// TIA Portal V16 export
// export: Created 2024-12-03T15:41:43.2889694Z, ExportSetting WithDefaults, DisplayName Totally Integrated Automation Portal, DisplayVersion V16 Update 6, DisplayName TIA Portal Version Control Interface, DisplayVersion V16 Update 2, DisplayName TIA Portal Openness, DisplayVersion V16 Update 6, DisplayName TIA Portal Teamcenter Gateway, DisplayVersion V16, DisplayName SINAMICS Startdrive Advanced, DisplayVersion V16 Update 5, DisplayName SINAMICS Startdrive G130, G150, S120, S150, SINAMICS MV, S210, DisplayVersion V16 Update 5, DisplayName SINAMICS Startdrive G110M, G120, G120C, G120D, G120P, G115D, DisplayVersion V16 Update 5, DisplayName STEP 7 Professional, DisplayVersion V16 Update 6, DisplayName STEP 7 Safety, DisplayVersion V16, DisplayName WinCC Advanced / Unified PC, DisplayVersion V16 Update 6
FUNCTION_BLOCK "Intersection_Controller_FB"   // FB30, SCL
{ S7_Optimized_Access := 'TRUE' }
VERSION : 0.1
// stored: AutoNumber true, IsIECCheckEnabled false, IsRetainMemResEnabled false, MemoryReserve 100, SetENOAutomatically false, UDAEnableTagReadback false
   VAR_INPUT
      I_con_upstream_north : Bool := TRUE;
      I_con_upstream_east : Bool := TRUE;
      I_con_upstream_south : Bool := TRUE;
      I_con_upstream_west : Bool := TRUE;
      I_Conv_North : "Conveyor_UDT";
      I_Conv_East : "Conveyor_UDT";
      I_Conv_South : "Conveyor_UDT";
      I_Conv_West : "Conveyor_UDT";
      I_Settings : "Intersection";
      I_AutoSent : Bool;
   END_VAR
   VAR_OUTPUT
      O_Empty_Flag : Bool;
   END_VAR
   VAR_IN_OUT
      IO_Conv_1 : "Conveyor_UDT";
      IO_Conv_2 : "Conveyor_UDT";
      IO_Transfer : "TransferUnitUpDown";
   END_VAR
   VAR
      Transfer : "ZPA_TransferUnit_Controller";
   END_VAR
   VAR RETAIN
      settings { S7_SetPoint := 'True'} : "Intersection";
   END_VAR
   VAR
      Empty { S7_SetPoint := 'True'} : "SmartBool";
   END_VAR
   VAR_TEMP
      T_Zone : "ZoneInfo";
      T_appstate : "ApplicationState_UDT";
      T_DownStream : "Conveyor_UDT";
      T_Upstream : "Conveyor_UDT";
      T_SendingConveyor : "Conveyor_UDT";
      T_ReceiveConveyor : "Conveyor_UDT";
      T_ReceivePosition : Int;
      T_InvalidSettings : Bool;
      T_Dummy : Bool;
      T_ConnectUpstream : Bool;
   END_VAR
BEGIN
   REGION INit temps

       #T_Zone := "ApplicationState_DB".ZoneNames[#IO_Conv_1.Zone];
       #T_appstate := "ApplicationState_DB".Appstate[#T_Zone.AppStateIndex];

       #T_DownStream := "CONV_DB".empty;
       #T_Upstream := "CONV_DB".empty;
       #T_SendingConveyor := "CONV_DB".empty;
       #T_ReceiveConveyor := "CONV_DB".empty;

   END_REGION

   REGION INIT NAMES

       IF #IO_Conv_1.Name = '' THEN
           #IO_Conv_1.Name := "buildObjectName"(I_Symbolname := GetSymbolName(variable:=#IO_Conv_1, size:=60));
       END_IF;

       IF #IO_Conv_2.Name = '' THEN
           #IO_Conv_2.Name := "buildObjectName"(I_Symbolname := GetSymbolName(variable := #IO_Conv_2, size := 60));
       END_IF;
   END_REGION

   REGION Allow new settings

       IF (#IO_Conv_1.Status.Empty
           AND #IO_Conv_2.Status.Empty) THEN //OR #settings.DownstreamIndex = 0 THEN
           #settings := #I_Settings;
       END_IF;

       #T_ReceivePosition := #settings.ReceivePosition;

   END_REGION

   REGION DownStream Selecotor

       CASE #settings.DownstreamIndex OF
           "North":
               #T_DownStream := #I_Conv_North  ;
           "East":
               #T_DownStream := #I_Conv_East ;
           "South":
               #T_DownStream := #I_Conv_South ;
           "West":
               #T_DownStream := #I_Conv_West ;
       END_CASE;

   END_REGION

   REGION Upstream selector

       #T_ConnectUpstream := FALSE;

       CASE #settings.UpstreamIndex OF
           "North":
               #T_Upstream := #I_Conv_North;
               #T_ConnectUpstream := #I_con_upstream_north;
           "East":
               #T_Upstream := #I_Conv_East;
               #T_ConnectUpstream := #I_con_upstream_east;
           "South":
               #T_Upstream := #I_Conv_South;
               #T_ConnectUpstream := #I_con_upstream_south;
           "West":
               #T_Upstream := #I_Conv_West;
               #T_ConnectUpstream := #I_con_upstream_west;
       END_CASE;

   END_REGION

   REGION Init conveyors

       #IO_Conv_1.Cmd.ReadyToReceive := 0;
       #IO_Conv_1.Cmd.ReadyToSent := 0;
       #IO_Conv_1.Cmd.InvertFlow := 0;
       #IO_Conv_1.Cmd.RunAuto := 0;

       #IO_Conv_1.Status.Empty := FALSE;

       #IO_Conv_1.Status.ExecutingReceiveSequence := FALSE;
       #IO_Conv_1.Status.ExecutingSendingSequence := FALSE;
       #IO_Conv_1.Status.RequestForSending := FALSE;

       #IO_Conv_2.Cmd.ReadyToReceive := 0;
       #IO_Conv_2.Cmd.ReadyToSent := 0;
       #IO_Conv_2.Cmd.InvertFlow := 0;
       #IO_Conv_2.Cmd.RunAuto := 0;

       #IO_Conv_2.Status.Empty := FALSE;

       #IO_Conv_2.Status.ExecutingReceiveSequence := FALSE;
       #IO_Conv_2.Status.ExecutingSendingSequence := FALSE;
       #IO_Conv_2.Status.RequestForSending := FALSE;

   END_REGION

   REGION Setup conveyors

       CASE #settings.ReceiveConveyorIndex OF
           1:
               #T_ReceiveConveyor := #IO_Conv_1;
           2:
               #T_ReceiveConveyor := #IO_Conv_2;
       END_CASE;

       CASE #settings.SendingConveyorIndex OF
           1:
               #T_SendingConveyor := #IO_Conv_1;
           2:
               #T_SendingConveyor := #IO_Conv_2;
       END_CASE;


       REGION ALIGNMENT OVERRIDE
           IF #Transfer.StepNumber = 60 THEN
               #T_ReceivePosition := #settings.Algin.AlginPosition;
               CASE #settings.Algin.conveyorIndex OF
                   1:
                       #T_ReceiveConveyor.Cmd := #IO_Conv_1.Cmd;
                       #T_ReceiveConveyor.Status := #IO_Conv_1.Status;
                       #T_ReceiveConveyor.Input := #IO_Conv_1.Input;
                       #T_ReceiveConveyor.Settings := #IO_Conv_1.Settings;
                       #T_ReceiveConveyor.Encoder := #IO_Conv_1.Encoder;
                   2:
                       #T_ReceiveConveyor.Cmd := #IO_Conv_2.Cmd;
                       #T_ReceiveConveyor.Status := #IO_Conv_2.Status;
                       #T_ReceiveConveyor.Input := #IO_Conv_2.Input;
                       #T_ReceiveConveyor.Settings := #IO_Conv_2.Settings;
                       #T_ReceiveConveyor.Encoder := #IO_Conv_2.Encoder;
               END_CASE;
           END_IF;
       END_REGION

       #T_ReceiveConveyor.Cmd.InvertFlow := #settings.InverseFlowReceiving;
       #T_SendingConveyor.Cmd.InvertFlow := #settings.InverseFlowSending;

   END_REGION

   REGION ZPA transfer unit
       #T_InvalidSettings := FALSE;
       IF #settings.DownstreamIndex = 0
           OR #settings.UpstreamIndex = 0
           OR #settings.SendingConveyorIndex = 0
           OR #settings.ReceiveConveyorIndex = 0
           OR #settings.ReceivePosition = 0
           OR #settings.SendingPosition = 0 THEN
           #T_InvalidSettings := true;
       END_IF;

       IF #T_InvalidSettings THEN
           #T_ReceiveConveyor := #IO_Conv_1;
           #T_SendingConveyor := #IO_Conv_2;
           #settings.ReceivePosition := "Down";
           #settings.SendingPosition := "Up";
       END_IF;

       #Transfer(I_BuildName:=FALSE,
                 I_SentAtEnd:= #I_AutoSent,
                 I_ConnectUpstream:= #T_ConnectUpstream,
                 I_UpstreamConveyor := #T_Upstream,
                 I_DownStreamConveyor := #T_DownStream,
                 I_ReceivePosition := #T_ReceivePosition,
                 I_SendingPosition := #settings.SendingPosition,
                 I_NoEndSensor:= #settings.ReceiveNoEndSensor,
                 I_AlignAfterReceive:=#settings.Algin.active,
                 I_AlignConveyorIndex := 1, // We always the the align conveyor the receive conveyor and set the receive conveyor,
                 I_AlignSpeed:=#settings.Algin.speed,
                 I_AlignDirection:=#settings.Algin.direction,
                 I_AlignDistance:=#settings.Algin.distnace,
                 I_AlignPostition:=#settings.Algin.AlginPosition,
                 IO_ReceiveConveyor := #T_ReceiveConveyor,
                 IO_SendingConveyor := #T_SendingConveyor,
                 IO_VLV_Transfer := #IO_Transfer); 

       #T_Dummy := #T_SendingConveyor.Cmd.Direction;

   END_REGION

   REGION update conveyors with transfer unit commands

       IF #settings.ReceiveConveyorIndex <> #settings.SendingConveyorIndex THEN

           CASE #settings.ReceiveConveyorIndex OF
               1:
                   #IO_Conv_1 := #T_ReceiveConveyor;
               2:
                   #IO_Conv_2 := #T_ReceiveConveyor;
           END_CASE;

           CASE #settings.SendingConveyorIndex OF
               1:
                   #IO_Conv_1 := #T_SendingConveyor;
               2:
                   #IO_Conv_2 := #T_SendingConveyor;
           END_CASE;

       ELSE

           IF #settings.ReceiveConveyorIndex = 1 AND #settings.SendingConveyorIndex = 1 THEN

               #IO_Conv_1.Cmd.RunAuto := #T_ReceiveConveyor.Cmd.RunAuto OR #T_SendingConveyor.Cmd.RunAuto;

               IF #T_ReceiveConveyor.Status.ExecutingReceiveSequence THEN
                   #IO_Conv_1 := #T_ReceiveConveyor;
               ELSIF #T_SendingConveyor.Status.ExecutingSendingSequence THEN
                   #IO_Conv_1 := #T_SendingConveyor;
               END_IF;
           END_IF;

           IF #settings.ReceiveConveyorIndex = 2 AND #settings.SendingConveyorIndex = 2 THEN

               #IO_Conv_2.Cmd.RunAuto := #T_ReceiveConveyor.Cmd.RunAuto OR #T_SendingConveyor.Cmd.RunAuto;

               IF #T_ReceiveConveyor.Status.ExecutingReceiveSequence THEN
                   #IO_Conv_2 := #T_ReceiveConveyor;
               ELSIF #T_SendingConveyor.Status.ExecutingSendingSequence THEN
                   #IO_Conv_2 := #T_SendingConveyor;
               END_IF;
           END_IF;

       END_IF;

       REGION ALIGNMENT FUNCTION
           IF #Transfer.StepNumber = 60 THEN
               CASE #settings.Algin.conveyorIndex OF
                   1:
                       #IO_Conv_1.Cmd := #T_ReceiveConveyor.Cmd;
                       #IO_Conv_1.Input := #T_ReceiveConveyor.Input;
                       #IO_Conv_1.Status := #T_ReceiveConveyor.Status;
                       #IO_Conv_1.Encoder :=#T_ReceiveConveyor.Encoder;
                       #IO_Conv_1.Settings := #T_ReceiveConveyor.Settings;
                       #IO_Conv_2.Cmd.RunAuto := 0;
                   2:
                       #IO_Conv_2.Cmd := #T_ReceiveConveyor.Cmd;
                       #IO_Conv_2.Cmd := #T_ReceiveConveyor.Cmd;
                       #IO_Conv_2.Input := #T_ReceiveConveyor.Input;
                       #IO_Conv_2.Status := #T_ReceiveConveyor.Status;
                       #IO_Conv_2.Encoder := #T_ReceiveConveyor.Encoder;
                       #IO_Conv_2.Settings := #T_ReceiveConveyor.Settings;
                       #IO_Conv_1.Cmd.RunAuto := 0;
               END_CASE;
           END_IF;
       END_REGION

       //Empty status of conveyors must always be the same
       #IO_Conv_1.Status.Empty := #T_SendingConveyor.Status.Empty OR #T_ReceiveConveyor.Status.Empty;
       #IO_Conv_2.Status.Empty := #T_SendingConveyor.Status.Empty OR #T_ReceiveConveyor.Status.Empty;



   END_REGION

   REGION ALARMS

       #IO_Conv_1.Alarms := #T_SendingConveyor.Alarms;

       #IO_Conv_1.Alarms.BlockedReceive.Active := #T_SendingConveyor.Alarms.BlockedReceive.Active
       OR #T_ReceiveConveyor.Alarms.BlockedReceive.Active;

       #IO_Conv_1.Alarms.BlockedSending.Active := #T_SendingConveyor.Alarms.BlockedSending.Active
       OR #T_ReceiveConveyor.Alarms.BlockedSending.Active;

       #IO_Conv_1.Alarms.ToClose.Active := #T_SendingConveyor.Alarms.ToClose.Active
       OR #T_ReceiveConveyor.Alarms.ToClose.Active;

       #IO_Conv_1.Alarms.ToLong.Active := #T_SendingConveyor.Alarms.ToLong.Active
       OR #T_ReceiveConveyor.Alarms.ToLong.Active;

       #IO_Conv_1.Alarms.ToSmall.Active := #T_SendingConveyor.Alarms.ToSmall.Active
       OR #T_ReceiveConveyor.Alarms.ToSmall.Active;

       #IO_Conv_1.Alarms.Status := #T_SendingConveyor.Alarms.Status
       OR #T_ReceiveConveyor.Alarms.Status;

       #IO_Conv_2.Alarms := #IO_Conv_1.Alarms;

   END_REGION

   REGION No interfacing on invalid settings

       IF #T_InvalidSettings THEN
           #IO_Conv_1.Cmd.RunAuto := FALSE;
           #IO_Conv_1.Cmd.ReadyToReceive := FALSE;
           #IO_Conv_1.Cmd.ReadyToSent := FALSE;
           #IO_Conv_2.Cmd.RunAuto := FALSE;
           #IO_Conv_2.Cmd.ReadyToReceive := FALSE;
           #IO_Conv_2.Cmd.ReadyToSent := FALSE;
       END_IF;

       IF #IO_Conv_1.Cmd.ReInitialize OR
           #IO_Conv_2.Cmd.ReInitialize THEN
           #Transfer.StepNumber := 10;
       END_IF;

       #IO_Conv_1.Cmd.ReInitialize := FALSE;
       #IO_Conv_2.Cmd.ReInitialize := FALSE;

   END_REGION

   REGION Clear settings on becoming empty

       #Empty(I_Sensor := #IO_Conv_1.Status.Empty);
       #O_Empty_Flag := #Empty.O_data.LE;
       IF #Empty.O_data.LE THEN
           #settings := "Intersection_DB".EmptySettings;
       END_IF;

   END_REGION
END_FUNCTION_BLOCK
